TYPE DataPositions :
STRUCT
	FeedInReadingPoint	:	WORD;
	FeedInStackerCrane	:	WORD;
	StackerCraneFork	:	WORD;
END_STRUCT
END_TYPE

(* stored: Version 1.1.0.1
   DUT DataPositions: Id {62d3f8c5-02f8-48fd-a0b0-c021127c544f} *)
